FUNCTION_BLOCK EL4028
VAR
	_io : EL4xx8_Data;
	{attribute addProperty Name "WcState"}
	_wcState : WcStateBase;
	{attribute addProperty Name "Info data"}
	_infoData : InfoDataAds;
END_VAR

PROPERTY IO : REFERENCE TO EL4xx8_Data
GET
IO REF= _io;
END_GET
END_PROPERTY

PROPERTY WcState : REFERENCE TO WcStateBase
GET
WcState REF= _wcState;
END_GET
END_PROPERTY

END_FUNCTION_BLOCK

(* stored: Version 1.1.0.1, ProductVersion 3.1.4024.9
   POU EL4028: Id {1b858de2-7da6-076e-08b9-207e915d495c}, SpecialFunc None
   Property IO: Id {a68d2f8e-36bd-02ce-338e-508449252f0a}
   Get Get: Id {bbbc3b88-25a1-08a9-30ad-4b2e7361fa8e}
   Property WcState: Id {3cc87d3f-0891-02f0-02f1-b33e9b8f4f44}
   Get Get: Id {0f7c2736-a8a6-0a5f-1d7f-0cfae0b37399} *)
